(* Schneider Machine Expert - Basic project magnetic-pulse-modbus, file version 2.5.0.0 *)
(* ProjectInformations: Name=AGM1-lower *)
(* UserInformations: LastName=Aleksandr, FirstName=Kolodkin, PhoneNumber=+380963724869, CellNumber=+380996102231, Email=alexandr.kolodkin@gmail.com *)

HARDWARE
  Cpu 0: TM221CE40T
  EthernetConfiguration: NetworkName=M221, IpAllocationMode=FixedAddress, IpAddress=192.168.10.21, SubnetMask=255.255.255.0
  SerialLineConfiguration: Baud=Baud19200, Parity=ParityEven, DataBits=DataBits8, StopBits=StopBits1, PhysicalMedium=PhysicalMediumRs485, TransmissionMode=TransmissionModeModbusRtu, SlaveId=1, Addressing=SlaveAddressing
  MastTask: UsePeriodScanMode=false, PeriodScan=100
  FastTask: Period=255
  CpuBehavior: StartingMode=StartInRun, AutoSaveRamOnEeprom=true, WatchdogPeriod=250

SYMBOLS  (address, symbol, comment, settings)
  %M0       INPUT_0  "Дискретный вход #0"
  %M1       INPUT_1  "Дискретный вход #1"
  %M2       INPUT_2  "Дискретный вход #2"
  %M3       INPUT_3  "Дискретный вход #3"
  %M4       INPUT_4  "Дискретный вход #4"
  %M5       INPUT_5  "Дискретный вход #5"
  %M6       INPUT_6  "Дискретный вход #6"
  %M7       INPUT_7  "Дискретный вход #7"
  %M8       INPUT_8  "Дискретный вход #8"
  %M9       INPUT_9  "Дискретный вход #9"
  %M10      INPUT_10  "Дискретный вход #10"
  %M11      INPUT_11  "Дискретный вход #11"
  %M12      INPUT_12  "Дискретный вход #12"
  %M13      INPUT_13  "Дискретный вход #13"
  %M14      INPUT_14  "Дискретный вход #14"
  %M15      INPUT_15  "Дискретный вход #15"
  %M16      INPUT_16  "Дискретный вход #16"
  %M17      INPUT_17  "Дискретный вход #17"
  %M18      INPUT_18  "Дискретный вход #18"
  %M19      INPUT_19  "Дискретный вход #19"
  %M20      INPUT_20  "Дискретный вход #20"
  %M21      INPUT_21  "Дискретный вход #21"
  %M22      INPUT_22  "Дискретный вход #22"
  %M23      INPUT_23  "Дискретный вход #23"
  %M24      INPUT_24  "Дискретный вход модуля расширения #0"
  %M25      INPUT_25  "Дискретный вход модуля расширения #1"
  %M26      INPUT_26  "Дискретный вход модуля расширения #2"
  %M27      INPUT_27  "Дискретный вход модуля расширения #3"
  %M28      INPUT_28  "Дискретный вход модуля расширения #4"
  %M29      INPUT_29  "Дискретный вход модуля расширения #5"
  %M30      INPUT_30  "Дискретный вход модуля расширения #6"
  %M31      INPUT_31  "Дискретный вход модуля расширения #7"
  %M32      LOCAL_1  "Местный запуск обрушения 1-го бункера"
  %M33      LOCAL_2  "Местный запуск обрушения 2-го бункера"
  %M34      LOCAL_3  "Местный запуск обрушения 3-го бункера"
  %M35      LOCAL_4  "Местный запуск обрушения 4-го бункера"
  %M36      LOCAL_5  "Местный запуск обрушения 5-го бункера"
  %M37      LOCAL_6  "Местный запуск обрушения 6-го бункера"
  %M38      LOCAL_7  "Местный запуск обрушения 7-го бункера"
  %M39      LOCAL_8  "Местный запуск обрушения 8-го бункера"
  %M40      LOCAL_9  "Местный запуск обрушения 9-го бункера"
  %M41      LOCAL_10  "Местный запуск обрушения 10-го бункера"
  %M48      REMOTE_1  "Дистанционный запуск обрушения 1-го бункера"
  %M49      REMOTE_2  "Дистанционный запуск обрушения 2-го бункера"
  %M50      REMOTE_3  "Дистанционный запуск обрушения 3-го бункера"
  %M51      REMOTE_4  "Дистанционный запуск обрушения 4-го бункера"
  %M52      REMOTE_5  "Дистанционный запуск обрушения 5-го бункера"
  %M53      REMOTE_6  "Дистанционный запуск обрушения 6-го бункера"
  %M54      REMOTE_7  "Дистанционный запуск обрушения 7-го бункера"
  %M55      REMOTE_8  "Дистанционный запуск обрушения 8-го бункера"
  %M56      REMOTE_9  "Дистанционный запуск обрушения 9-го бункера"
  %M57      REMOTE_10  "Дистанционный запуск обрушения 10-го бункера"
  %M64      CMD_1  "Заказано обрушение 1-го бункера"
  %M65      CMD_2  "Заказано обрушение 2-го бункера"
  %M66      CMD_3  "Заказано обрушение 3-го бункера"
  %M67      CMD_4  "Заказано обрушение 4-го бункера"
  %M68      CMD_5  "Заказано обрушение 5-го бункера"
  %M69      CMD_6  "Заказано обрушение 6-го бункера"
  %M70      CMD_7  "Заказано обрушение 7-го бункера"
  %M71      CMD_8  "Заказано обрушение 8-го бункера"
  %M72      CMD_9  "Заказано обрушение 9-го бункера"
  %M73      CMD_10  "Заказано обрушение 10-го бункера"
  %M80      CMD  "Есть заказ на обрушение бункера"
  %M81      RESET  "Сброс"
  %M82      READY  "Готовность"
  %M83      FAULT  "Авария при заряде конденсатора"
  %M84      TEMP  "Промежуточная переменная для получения сигнала NEXT"
  %M85      PULSE  "Импульс"
  %M86      NEXT  "Переход к следующему заказу или завершение работы"
  %M87      CHARGED  "Конденсатор заряжен"
  %M88      LOCAL  "Выбрано местное управление"
  %M89      REMOTE  "Выбрано дистанционное управление"
  %M90      POWER  "Питание подано"
  %M91      CHARGE  "Комманда на заряд конденсатора"
  %M96      PULSE_1  "Запуск обрушения 1-го бункера"
  %M97      PULSE_2  "Запуск обрушения 2-го бункера"
  %M98      PULSE_3  "Запуск обрушения 3-го бункера"
  %M99      PULSE_4  "Запуск обрушения 4-го бункера"
  %M100     PULSE_5  "Запуск обрушения 5-го бункера"
  %M101     PULSE_6  "Запуск обрушения 6-го бункера"
  %M102     PULSE_7  "Запуск обрушения 7-го бункера"
  %M103     PULSE_8  "Запуск обрушения 8-го бункера"
  %M104     PULSE_9  "Запуск обрушения 9-го бункера"
  %M105     PULSE_10  "Запуск обрушения 10-го бункера"
  %M112     SELECTED_1  "Выполняется обрушение 1-го бункера"
  %M113     SELECTED_2  "Выполняется обрушение 2-го бункера"
  %M114     SELECTED_3  "Выполняется обрушение 3-го бункера"
  %M115     SELECTED_4  "Выполняется обрушение 4-го бункера"
  %M116     SELECTED_5  "Выполняется обрушение 5-го бункера"
  %M117     SELECTED_6  "Выполняется обрушение 6-го бункера"
  %M118     SELECTED_7  "Выполняется обрушение 7-го бункера"
  %M119     SELECTED_8  "Выполняется обрушение 8-го бункера"
  %M120     SELECTED_9  "Выполняется обрушение 9-го бункера"
  %M121     SELECTED_10  "Выполняется обрушение 10-го бункера"
  %M128     MODBUS_1  "Запуск обрушения 1-го бункера через ModBus"
  %M129     MODBUS_2  "Запуск обрушения 2-го бункера через ModBus"
  %M130     MODBUS_3  "Запуск обрушения 3-го бункера через ModBus"
  %M131     MODBUS_4  "Запуск обрушения 4-го бункера через ModBus"
  %M132     MODBUS_5  "Запуск обрушения 5-го бункера через ModBus"
  %M133     MODBUS_6  "Запуск обрушения 6-го бункера через ModBus"
  %M134     MODBUS_7  "Запуск обрушения 7-го бункера через ModBus"
  %M135     MODBUS_8  "Запуск обрушения 8-го бункера через ModBus"
  %M136     MODBUS_9  "Запуск обрушения 9-го бункера через ModBus"
  %M137     MODBUS_10  "Запуск обрушения 10-го бункера через ModBus"
  %M144     MODBUS  "Управление по сети ModBus"
  %M145     CHARGED_M  "Имитация конденсатора при управлении по ModBus'у"
  %M146     RESET_M  "Сброс аварии по сети ModBus"
  %M160     FAULT_1  "Сбой при обрушении 1-го бункера"
  %M161     FAULT_2  "Сбой при обрушении 2-го бункера"
  %M162     FAULT_3  "Сбой при обрушении 3-го бункера"
  %M163     FAULT_4  "Сбой при обрушении 4-го бункера"
  %M164     FAULT_5  "Сбой при обрушении 5-го бункера"
  %M165     FAULT_6  "Сбой при обрушении 6-го бункера"
  %M166     FAULT_7  "Сбой при обрушении 7-го бункера"
  %M167     FAULT_8  "Сбой при обрушении 8-го бункера"
  %M168     FAULT_9  "Сбой при обрушении 9-го бункера"
  %M169     FAULT_10  "Сбой при обрушении 10-го бункера"
  %TM0      READY_T  "Задержка готовности"  [Preset=10, Base=OneHundredMilliSeconds]
  %TM1      RESET_T  "Импульс сброса"  [Type=TOF, Preset=5, Base=OneHundredMilliSeconds]
  %TM2      CHARGE_T  "Задержка начала заряда конденсатора"  [Preset=10, Base=TenMilliSeconds]
  %TM3      CHARGE_FAULT_T  "Задержка до аварии: конденсатор не заряжен"  [Preset=15, Base=OneSecond]
  %TM4      DISCHARGE_FAULT_T  "Задержка до аварии: конденсатор не разряжен"  [Preset=30, Base=OneHundredMilliSeconds]
  %TM5      PULSE_START_T  "Задержка перед подачей импульса"  [Preset=20, Base=OneHundredMilliSeconds]
  %TM6      PULSE_T  "Продолжительность импульса"  [Type=TP, Preset=50, Base=TenMilliSeconds]
  %TM7      NEXT_T  "Задержка перед началом проверки (должно быть меньше чем DISCHARGE_FAULT_T)"  [Type=TOF, Preset=5, Base=OneHundredMilliSeconds]
  %TM10     CMD1_T  "Формирование имульса заказа #1"  [Type=TP, Preset=1, Base=TenMilliSeconds]
  %TM11     CMD2_T  "Формирование имульса заказа #2"  [Type=TP, Preset=1, Base=TenMilliSeconds]
  %TM12     CMD3_T  "Формирование имульса заказа #3"  [Type=TP, Preset=1, Base=TenMilliSeconds]
  %TM13     CMD4_T  "Формирование имульса заказа #4"  [Type=TP, Preset=1, Base=TenMilliSeconds]
  %TM14     CMD5_T  "Формирование имульса заказа #5"  [Type=TP, Preset=1, Base=TenMilliSeconds]
  %TM15     CMD6_T  "Формирование имульса заказа #6"  [Type=TP, Preset=1, Base=TenMilliSeconds]
  %TM16     CMD7_T  "Формирование имульса заказа #7"  [Type=TP, Preset=1, Base=TenMilliSeconds]
  %TM17     CMD8_T  "Формирование имульса заказа #8"  [Type=TP, Preset=1, Base=TenMilliSeconds]
  %READ_VAR0 RD3_1  [Link(Value(FBComLinkParameterEnums=SerialLine1)), RemoteDeviceId(Value(int=1)), Timeout(Value(int=100)), ObjType(Value(FBComObjTypeParameterEnums=MW)), FirstObj(Value(int=0)), Quantity(Value(int=16)), IndexData(Value(int=0))]
  %I0.0     IN_0
  %I0.1     IN_1
  %I0.2     IN_2
  %I0.3     IN_3
  %I0.4     IN_4
  %I0.5     IN_5
  %I0.6     IN_6
  %I0.7     IN_7
  %I0.8     IN_8
  %I0.9     IN_9
  %I0.10    IN_10
  %I0.11    IN_11
  %I0.12    IN_12
  %I0.13    IN_13
  %I0.14    IN_14
  %I0.15    IN_15
  %I0.16    IN_16
  %I0.17    IN_17
  %I0.18    IN_18
  %I0.19    IN_19
  %I0.20    IN_20
  %I0.21    IN_21
  %I0.22    IN_22
  %I0.23    IN_23
  %Q0.0     OUTPUT_0
  %Q0.1     OUTPUT_1  "Запуск №2"
  %Q0.2     OUTPUT_2  "Запуск №3"
  %Q0.3     OUTPUT_3  "Запуск №4"
  %Q0.4     OUTPUT_4  "Запуск №5"
  %Q0.5     OUTPUT_5  "Запуск №6"
  %Q0.6     OUTPUT_6  "Запуск №7"
  %Q0.7     OUTPUT_7  "Запуск №8"
  %Q0.8     OUTPUT_8
  %Q0.9     OUTPUT_9
  %Q0.10    OUTPUT_10  "Готовность"
  %Q0.11    OUTPUT_11
  %Q0.12    OUTPUT_12
  %Q0.13    OUTPUT_13
  %Q0.14    OUTPUT_14  "Включить заряд конденсатора"
  %Q0.15    OUTPUT_15  "Ошибка"

POU Main logic
  (* SectionNumber=1 *)

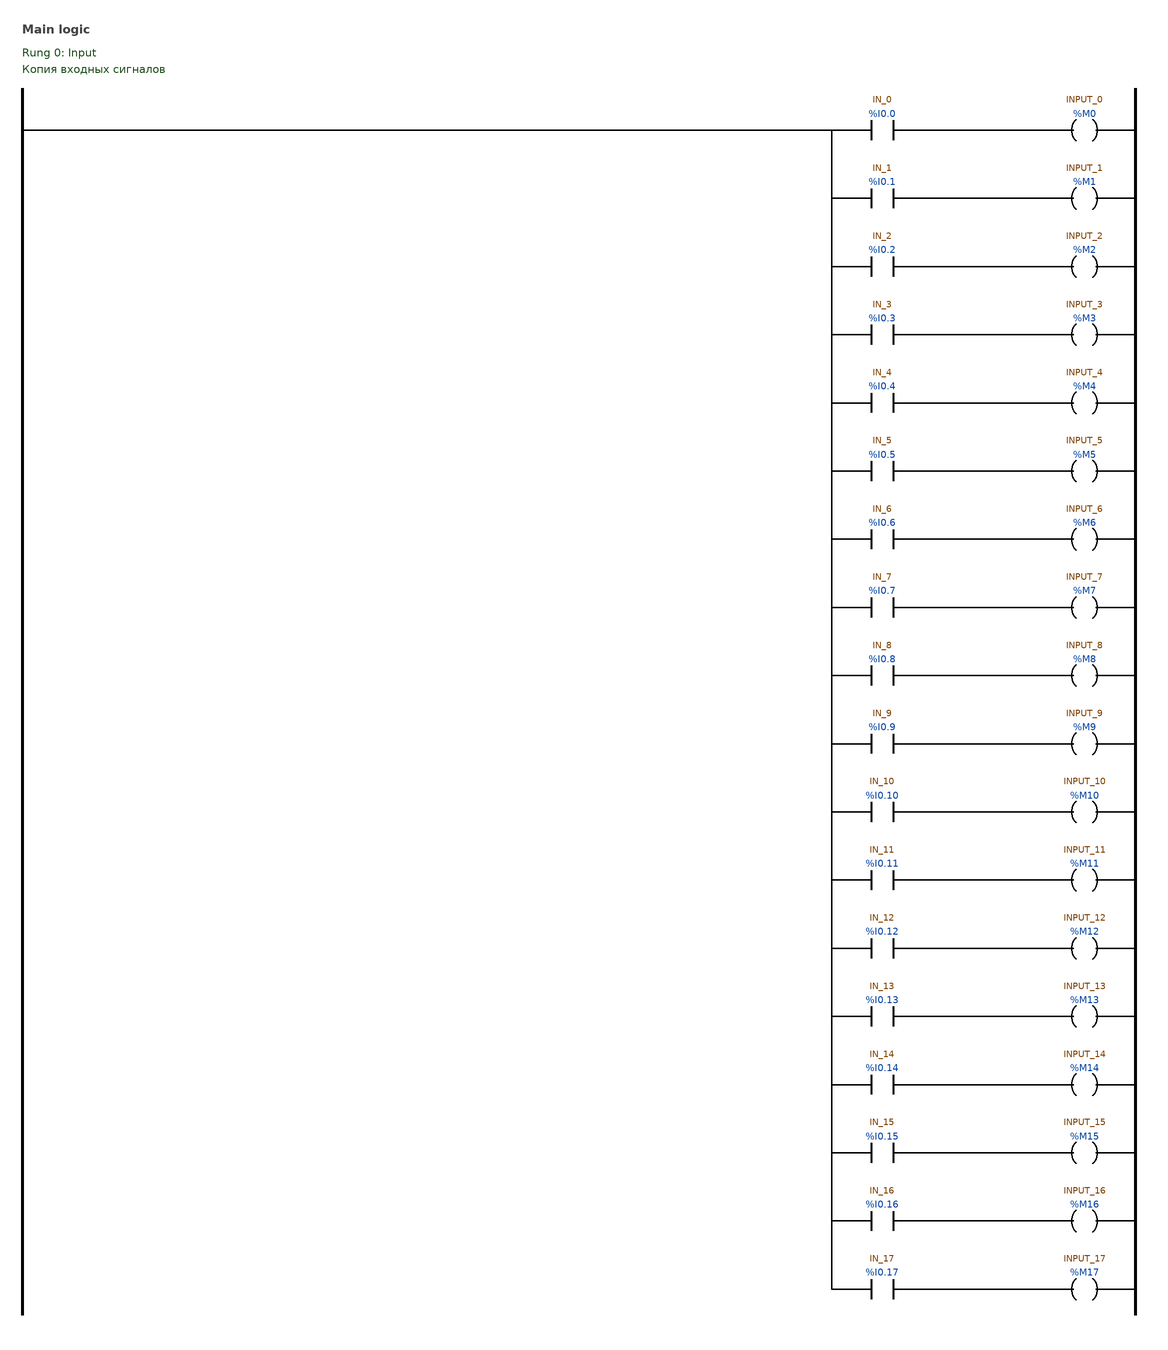

// Rung 0: Input
// Копия входных сигналов
  LD 1
  MPS
  AND %I0.0               (* IN_0 *)
  ST %M0                  (* INPUT_0 *)
  MRD
  AND %I0.1               (* IN_1 *)
  ST %M1                  (* INPUT_1 *)
  MRD
  AND %I0.2               (* IN_2 *)
  ST %M2                  (* INPUT_2 *)
  MRD
  AND %I0.3               (* IN_3 *)
  ST %M3                  (* INPUT_3 *)
  MRD
  AND %I0.4               (* IN_4 *)
  ST %M4                  (* INPUT_4 *)
  MRD
  AND %I0.5               (* IN_5 *)
  ST %M5                  (* INPUT_5 *)
  MRD
  AND %I0.6               (* IN_6 *)
  ST %M6                  (* INPUT_6 *)
  MRD
  AND %I0.7               (* IN_7 *)
  ST %M7                  (* INPUT_7 *)
  MRD
  AND %I0.8               (* IN_8 *)
  ST %M8                  (* INPUT_8 *)
  MRD
  AND %I0.9               (* IN_9 *)
  ST %M9                  (* INPUT_9 *)
  MRD
  AND %I0.10              (* IN_10 *)
  ST %M10                 (* INPUT_10 *)
  MRD
  AND %I0.11              (* IN_11 *)
  ST %M11                 (* INPUT_11 *)
  MRD
  AND %I0.12              (* IN_12 *)
  ST %M12                 (* INPUT_12 *)
  MRD
  AND %I0.13              (* IN_13 *)
  ST %M13                 (* INPUT_13 *)
  MRD
  AND %I0.14              (* IN_14 *)
  ST %M14                 (* INPUT_14 *)
  MRD
  AND %I0.15              (* IN_15 *)
  ST %M15                 (* INPUT_15 *)
  MRD
  AND %I0.16              (* IN_16 *)
  ST %M16                 (* INPUT_16 *)
  MPP
  AND %I0.17              (* IN_17 *)
  ST %M17                 (* INPUT_17 *)
  // as ST:
  //   INPUT_0 := IN_0;
  //   INPUT_1 := IN_1;
  //   INPUT_2 := IN_2;
  //   INPUT_3 := IN_3;
  //   INPUT_4 := IN_4;
  //   INPUT_5 := IN_5;
  //   INPUT_6 := IN_6;
  //   INPUT_7 := IN_7;
  //   INPUT_8 := IN_8;
  //   INPUT_9 := IN_9;
  //   INPUT_10 := IN_10;
  //   INPUT_11 := IN_11;
  //   INPUT_12 := IN_12;
  //   INPUT_13 := IN_13;
  //   INPUT_14 := IN_14;
  //   INPUT_15 := IN_15;
  //   INPUT_16 := IN_16;
  //   INPUT_17 := IN_17;

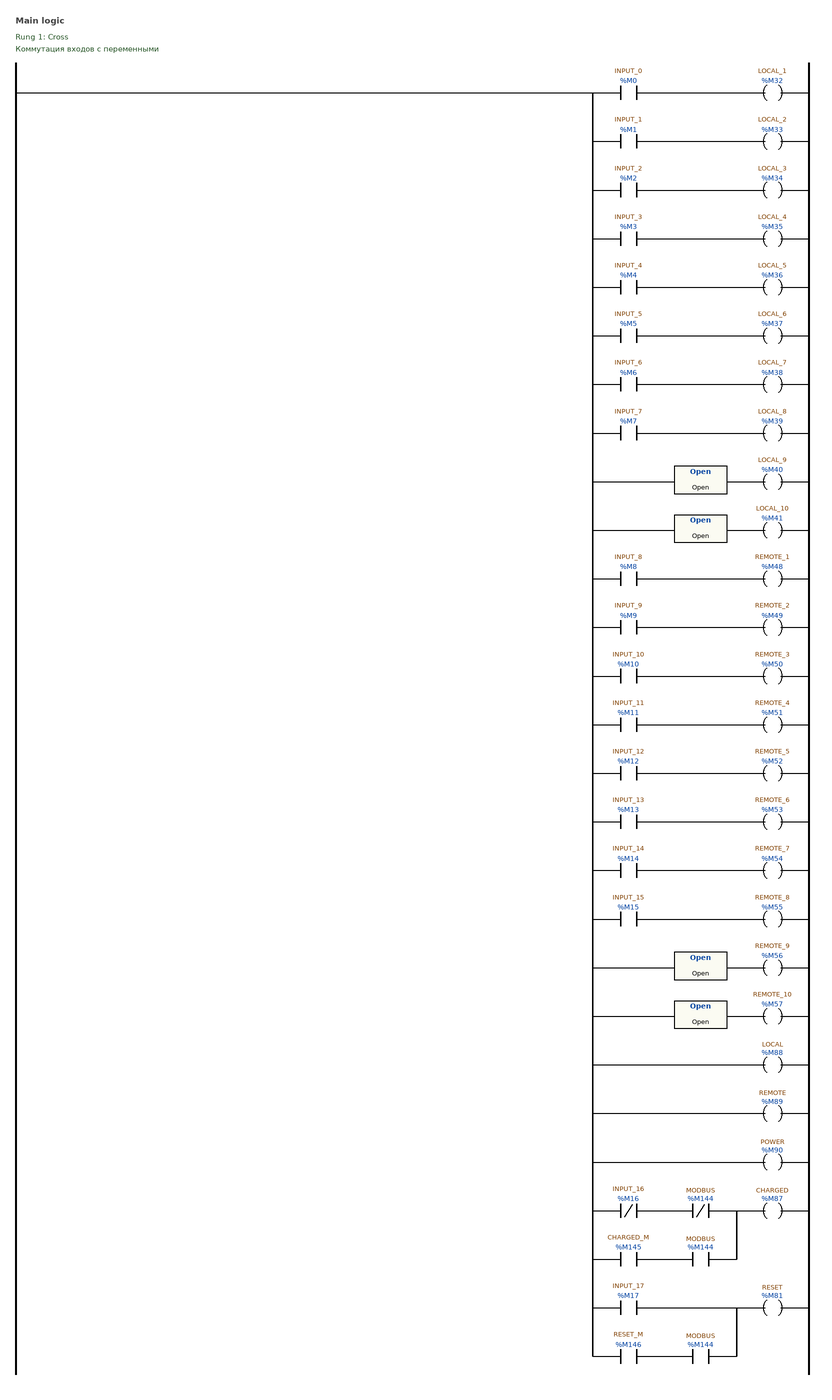

// Rung 1: Cross
// Коммутация входов с переменными
  LD 1
  MPS
  AND %M0                 (* INPUT_0 *)
  ST %M32                 (* LOCAL_1 *)
  MRD
  AND %M1                 (* INPUT_1 *)
  ST %M33                 (* LOCAL_2 *)
  MRD
  AND %M2                 (* INPUT_2 *)
  ST %M34                 (* LOCAL_3 *)
  MRD
  AND %M3                 (* INPUT_3 *)
  ST %M35                 (* LOCAL_4 *)
  MRD
  AND %M4                 (* INPUT_4 *)
  ST %M36                 (* LOCAL_5 *)
  MRD
  AND %M5                 (* INPUT_5 *)
  ST %M37                 (* LOCAL_6 *)
  MRD
  AND %M6                 (* INPUT_6 *)
  ST %M38                 (* LOCAL_7 *)
  MRD
  AND %M7                 (* INPUT_7 *)
  ST %M39                 (* LOCAL_8 *)
  MRD
  AND 0
  ST %M40                 (* LOCAL_9 *)
  MRD
  AND 0
  ST %M41                 (* LOCAL_10 *)
  MRD
  AND %M8                 (* INPUT_8 *)
  ST %M48                 (* REMOTE_1 *)
  MRD
  AND %M9                 (* INPUT_9 *)
  ST %M49                 (* REMOTE_2 *)
  MRD
  AND %M10                (* INPUT_10 *)
  ST %M50                 (* REMOTE_3 *)
  MRD
  AND %M11                (* INPUT_11 *)
  ST %M51                 (* REMOTE_4 *)
  MRD
  AND %M12                (* INPUT_12 *)
  ST %M52                 (* REMOTE_5 *)
  MRD
  AND %M13                (* INPUT_13 *)
  ST %M53                 (* REMOTE_6 *)
  MRD
  AND %M14                (* INPUT_14 *)
  ST %M54                 (* REMOTE_7 *)
  MRD
  AND %M15                (* INPUT_15 *)
  ST %M55                 (* REMOTE_8 *)
  MRD
  AND 0
  ST %M56                 (* REMOTE_9 *)
  MRD
  AND 0
  ST %M57                 (* REMOTE_10 *)
  MRD
  AND 1
  ST %M88                 (* LOCAL *)
  MRD
  AND 1
  ST %M89                 (* REMOTE *)
  MRD
  AND 1
  ST %M90                 (* POWER *)
  MRD
  AND(N %M16              (* INPUT_16 *)
  ANDN %M144              (* MODBUS *)
  OR( %M145               (* CHARGED_M *)
  AND %M144               (* MODBUS *)
  )
  )
  ST %M87                 (* CHARGED *)
  MPP
  AND( %M17               (* INPUT_17 *)
  OR( %M146               (* RESET_M *)
  AND %M144               (* MODBUS *)
  )
  )
  ST %M81                 (* RESET *)
  // as ST:
  //   LOCAL_1 := INPUT_0;
  //   LOCAL_2 := INPUT_1;
  //   LOCAL_3 := INPUT_2;
  //   LOCAL_4 := INPUT_3;
  //   LOCAL_5 := INPUT_4;
  //   LOCAL_6 := INPUT_5;
  //   LOCAL_7 := INPUT_6;
  //   LOCAL_8 := INPUT_7;
  //   LOCAL_9 := FALSE;
  //   LOCAL_10 := FALSE;
  //   REMOTE_1 := INPUT_8;
  //   REMOTE_2 := INPUT_9;
  //   REMOTE_3 := INPUT_10;
  //   REMOTE_4 := INPUT_11;
  //   REMOTE_5 := INPUT_12;
  //   REMOTE_6 := INPUT_13;
  //   REMOTE_7 := INPUT_14;
  //   REMOTE_8 := INPUT_15;
  //   REMOTE_9 := FALSE;
  //   REMOTE_10 := FALSE;
  //   LOCAL := TRUE;
  //   REMOTE := TRUE;
  //   POWER := TRUE;
  //   CHARGED := NOT INPUT_16 AND NOT MODBUS OR CHARGED_M AND MODBUS;
  //   RESET := INPUT_17 OR RESET_M AND MODBUS;

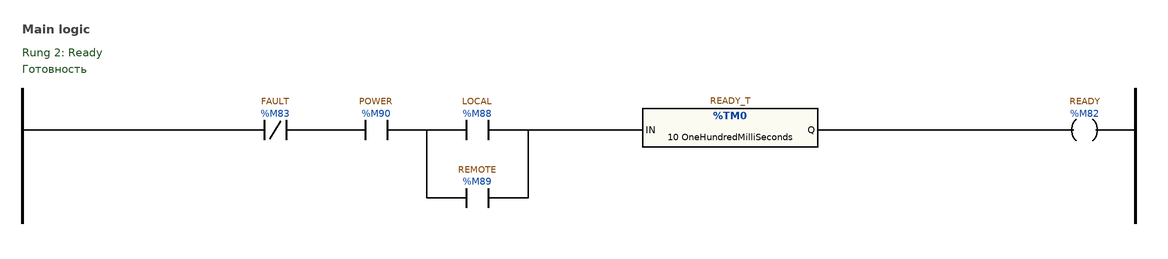

// Rung 2: Ready
// Готовность
  BLK %TM0                (* READY_T *)
  LDN %M83                (* FAULT *)
  AND %M90                (* POWER *)
  AND( %M88               (* LOCAL *)
  OR %M89                 (* REMOTE *)
  )
  IN
  OUT_BLK
  LD Q
  ST %M82                 (* READY *)
  END_BLK
  // as ST:
  //   READY_T(IN := NOT FAULT AND POWER AND (LOCAL OR REMOTE));
  //   READY := READY_T.Q;

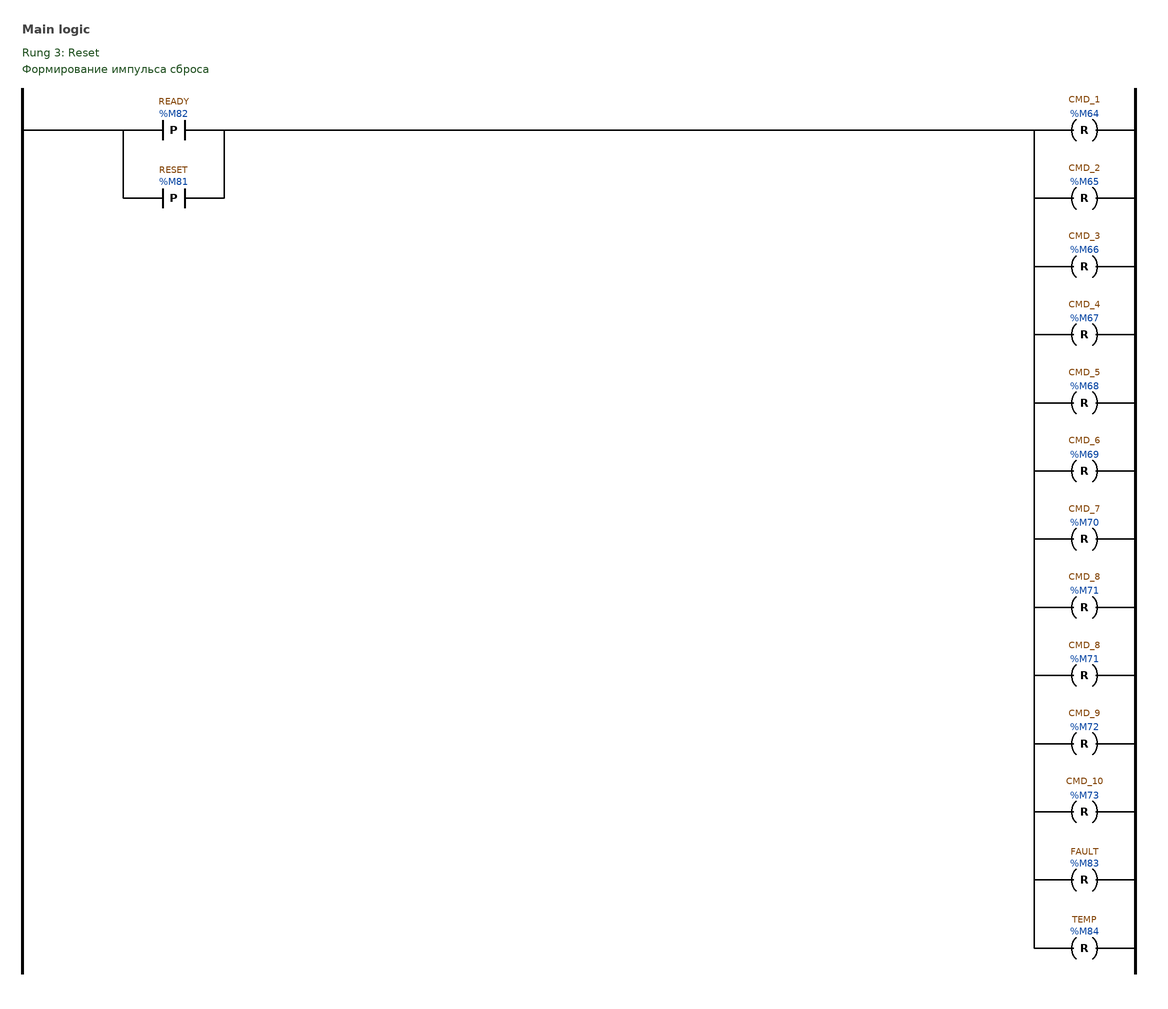

// Rung 3: Reset
// Формирование импульса сброса
  LD 1
  AND(R %M82              (* READY *)
  ORR %M81                (* RESET *)
  )
  R %M64                  (* CMD_1 *)
  R %M65                  (* CMD_2 *)
  R %M66                  (* CMD_3 *)
  R %M67                  (* CMD_4 *)
  R %M68                  (* CMD_5 *)
  R %M69                  (* CMD_6 *)
  R %M70                  (* CMD_7 *)
  R %M71                  (* CMD_8 *)
  R %M71                  (* CMD_8 *)
  R %M72                  (* CMD_9 *)
  R %M73                  (* CMD_10 *)
  R %M83                  (* FAULT *)
  R %M84                  (* TEMP *)
  // as ST:
  //   IF RISING(READY) OR RISING(RESET) THEN CMD_1 := FALSE; END_IF;
  //   IF RISING(READY) OR RISING(RESET) THEN CMD_2 := FALSE; END_IF;
  //   IF RISING(READY) OR RISING(RESET) THEN CMD_3 := FALSE; END_IF;
  //   IF RISING(READY) OR RISING(RESET) THEN CMD_4 := FALSE; END_IF;
  //   IF RISING(READY) OR RISING(RESET) THEN CMD_5 := FALSE; END_IF;
  //   IF RISING(READY) OR RISING(RESET) THEN CMD_6 := FALSE; END_IF;
  //   IF RISING(READY) OR RISING(RESET) THEN CMD_7 := FALSE; END_IF;
  //   IF RISING(READY) OR RISING(RESET) THEN CMD_8 := FALSE; END_IF;
  //   IF RISING(READY) OR RISING(RESET) THEN CMD_8 := FALSE; END_IF;
  //   IF RISING(READY) OR RISING(RESET) THEN CMD_9 := FALSE; END_IF;
  //   IF RISING(READY) OR RISING(RESET) THEN CMD_10 := FALSE; END_IF;
  //   IF RISING(READY) OR RISING(RESET) THEN FAULT := FALSE; END_IF;
  //   IF RISING(READY) OR RISING(RESET) THEN TEMP := FALSE; END_IF;

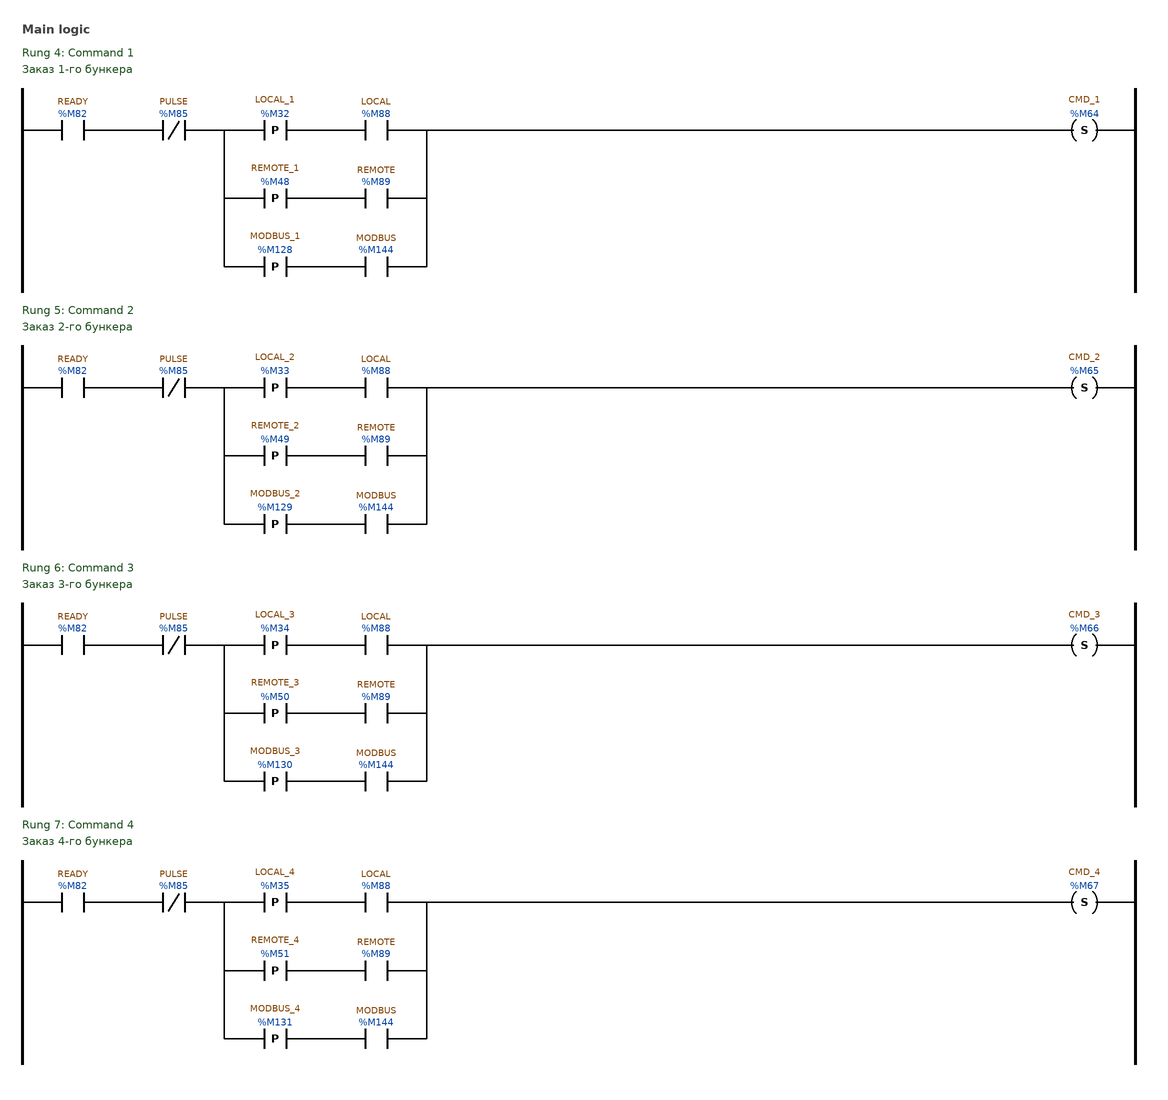

// Rung 4: Command 1
// Заказ 1-го бункера
  LD %M82                 (* READY *)
  ANDN %M85               (* PULSE *)
  AND(R %M32              (* LOCAL_1 *)
  AND %M88                (* LOCAL *)
  OR(R %M48               (* REMOTE_1 *)
  AND %M89                (* REMOTE *)
  )
  OR(R %M128              (* MODBUS_1 *)
  AND %M144               (* MODBUS *)
  )
  )
  S %M64                  (* CMD_1 *)
  // as ST:
  //   IF READY AND NOT PULSE AND (RISING(LOCAL_1) AND LOCAL OR RISING(REMOTE_1) AND REMOTE OR RISING(MODBUS_1) AND MODBUS) THEN CMD_1 := TRUE; END_IF;

// Rung 5: Command 2
// Заказ 2-го бункера
  LD %M82                 (* READY *)
  ANDN %M85               (* PULSE *)
  AND(R %M33              (* LOCAL_2 *)
  AND %M88                (* LOCAL *)
  OR(R %M49               (* REMOTE_2 *)
  AND %M89                (* REMOTE *)
  )
  OR(R %M129              (* MODBUS_2 *)
  AND %M144               (* MODBUS *)
  )
  )
  S %M65                  (* CMD_2 *)
  // as ST:
  //   IF READY AND NOT PULSE AND (RISING(LOCAL_2) AND LOCAL OR RISING(REMOTE_2) AND REMOTE OR RISING(MODBUS_2) AND MODBUS) THEN CMD_2 := TRUE; END_IF;

// Rung 6: Command 3
// Заказ 3-го бункера
  LD %M82                 (* READY *)
  ANDN %M85               (* PULSE *)
  AND(R %M34              (* LOCAL_3 *)
  AND %M88                (* LOCAL *)
  OR(R %M50               (* REMOTE_3 *)
  AND %M89                (* REMOTE *)
  )
  OR(R %M130              (* MODBUS_3 *)
  AND %M144               (* MODBUS *)
  )
  )
  S %M66                  (* CMD_3 *)
  // as ST:
  //   IF READY AND NOT PULSE AND (RISING(LOCAL_3) AND LOCAL OR RISING(REMOTE_3) AND REMOTE OR RISING(MODBUS_3) AND MODBUS) THEN CMD_3 := TRUE; END_IF;

// Rung 7: Command 4
// Заказ 4-го бункера
  LD %M82                 (* READY *)
  ANDN %M85               (* PULSE *)
  AND(R %M35              (* LOCAL_4 *)
  AND %M88                (* LOCAL *)
  OR(R %M51               (* REMOTE_4 *)
  AND %M89                (* REMOTE *)
  )
  OR(R %M131              (* MODBUS_4 *)
  AND %M144               (* MODBUS *)
  )
  )
  S %M67                  (* CMD_4 *)
  // as ST:
  //   IF READY AND NOT PULSE AND (RISING(LOCAL_4) AND LOCAL OR RISING(REMOTE_4) AND REMOTE OR RISING(MODBUS_4) AND MODBUS) THEN CMD_4 := TRUE; END_IF;

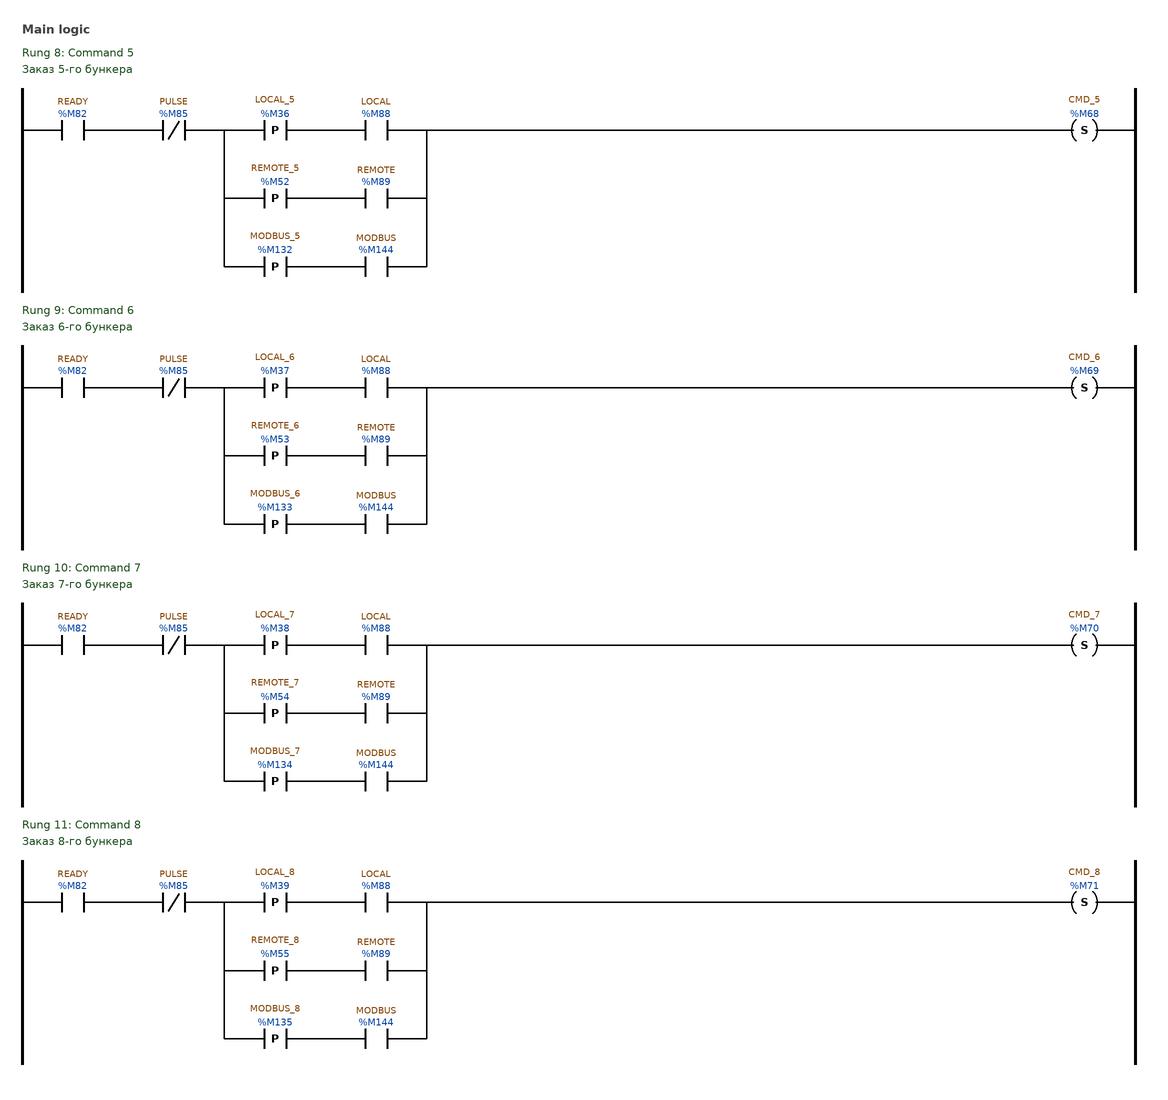

// Rung 8: Command 5
// Заказ 5-го бункера
  LD %M82                 (* READY *)
  ANDN %M85               (* PULSE *)
  AND(R %M36              (* LOCAL_5 *)
  AND %M88                (* LOCAL *)
  OR(R %M52               (* REMOTE_5 *)
  AND %M89                (* REMOTE *)
  )
  OR(R %M132              (* MODBUS_5 *)
  AND %M144               (* MODBUS *)
  )
  )
  S %M68                  (* CMD_5 *)
  // as ST:
  //   IF READY AND NOT PULSE AND (RISING(LOCAL_5) AND LOCAL OR RISING(REMOTE_5) AND REMOTE OR RISING(MODBUS_5) AND MODBUS) THEN CMD_5 := TRUE; END_IF;

// Rung 9: Command 6
// Заказ 6-го бункера
  LD %M82                 (* READY *)
  ANDN %M85               (* PULSE *)
  AND(R %M37              (* LOCAL_6 *)
  AND %M88                (* LOCAL *)
  OR(R %M53               (* REMOTE_6 *)
  AND %M89                (* REMOTE *)
  )
  OR(R %M133              (* MODBUS_6 *)
  AND %M144               (* MODBUS *)
  )
  )
  S %M69                  (* CMD_6 *)
  // as ST:
  //   IF READY AND NOT PULSE AND (RISING(LOCAL_6) AND LOCAL OR RISING(REMOTE_6) AND REMOTE OR RISING(MODBUS_6) AND MODBUS) THEN CMD_6 := TRUE; END_IF;

// Rung 10: Command 7
// Заказ 7-го бункера
  LD %M82                 (* READY *)
  ANDN %M85               (* PULSE *)
  AND(R %M38              (* LOCAL_7 *)
  AND %M88                (* LOCAL *)
  OR(R %M54               (* REMOTE_7 *)
  AND %M89                (* REMOTE *)
  )
  OR(R %M134              (* MODBUS_7 *)
  AND %M144               (* MODBUS *)
  )
  )
  S %M70                  (* CMD_7 *)
  // as ST:
  //   IF READY AND NOT PULSE AND (RISING(LOCAL_7) AND LOCAL OR RISING(REMOTE_7) AND REMOTE OR RISING(MODBUS_7) AND MODBUS) THEN CMD_7 := TRUE; END_IF;

// Rung 11: Command 8
// Заказ 8-го бункера
  LD %M82                 (* READY *)
  ANDN %M85               (* PULSE *)
  AND(R %M39              (* LOCAL_8 *)
  AND %M88                (* LOCAL *)
  OR(R %M55               (* REMOTE_8 *)
  AND %M89                (* REMOTE *)
  )
  OR(R %M135              (* MODBUS_8 *)
  AND %M144               (* MODBUS *)
  )
  )
  S %M71                  (* CMD_8 *)
  // as ST:
  //   IF READY AND NOT PULSE AND (RISING(LOCAL_8) AND LOCAL OR RISING(REMOTE_8) AND REMOTE OR RISING(MODBUS_8) AND MODBUS) THEN CMD_8 := TRUE; END_IF;

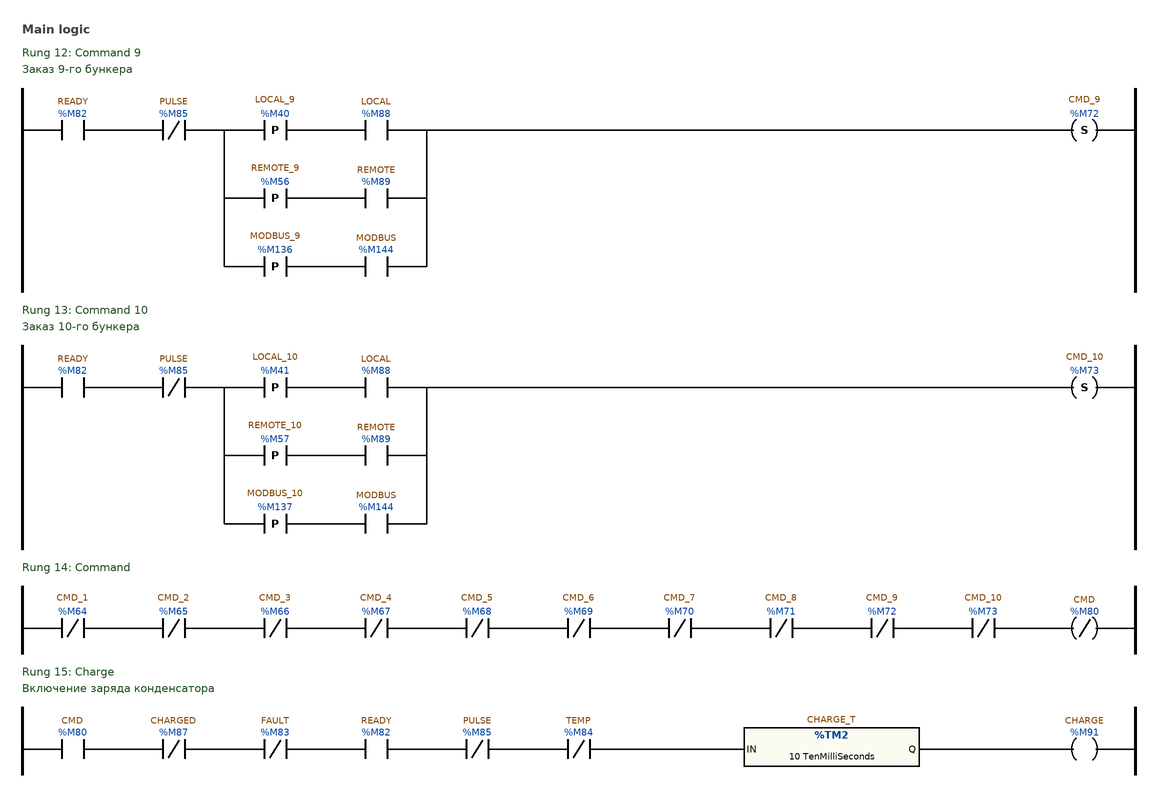

// Rung 12: Command 9
// Заказ 9-го бункера
  LD %M82                 (* READY *)
  ANDN %M85               (* PULSE *)
  AND(R %M40              (* LOCAL_9 *)
  AND %M88                (* LOCAL *)
  OR(R %M56               (* REMOTE_9 *)
  AND %M89                (* REMOTE *)
  )
  OR(R %M136              (* MODBUS_9 *)
  AND %M144               (* MODBUS *)
  )
  )
  S %M72                  (* CMD_9 *)
  // as ST:
  //   IF READY AND NOT PULSE AND (RISING(LOCAL_9) AND LOCAL OR RISING(REMOTE_9) AND REMOTE OR RISING(MODBUS_9) AND MODBUS) THEN CMD_9 := TRUE; END_IF;

// Rung 13: Command 10
// Заказ 10-го бункера
  LD %M82                 (* READY *)
  ANDN %M85               (* PULSE *)
  AND(R %M41              (* LOCAL_10 *)
  AND %M88                (* LOCAL *)
  OR(R %M57               (* REMOTE_10 *)
  AND %M89                (* REMOTE *)
  )
  OR(R %M137              (* MODBUS_10 *)
  AND %M144               (* MODBUS *)
  )
  )
  S %M73                  (* CMD_10 *)
  // as ST:
  //   IF READY AND NOT PULSE AND (RISING(LOCAL_10) AND LOCAL OR RISING(REMOTE_10) AND REMOTE OR RISING(MODBUS_10) AND MODBUS) THEN CMD_10 := TRUE; END_IF;

// Rung 14: Command
  LDN %M64                (* CMD_1 *)
  ANDN %M65               (* CMD_2 *)
  ANDN %M66               (* CMD_3 *)
  ANDN %M67               (* CMD_4 *)
  ANDN %M68               (* CMD_5 *)
  ANDN %M69               (* CMD_6 *)
  ANDN %M70               (* CMD_7 *)
  ANDN %M71               (* CMD_8 *)
  ANDN %M72               (* CMD_9 *)
  ANDN %M73               (* CMD_10 *)
  STN %M80                (* CMD *)
  // as ST:
  //   CMD := NOT (NOT CMD_1 AND NOT CMD_2 AND NOT CMD_3 AND NOT CMD_4 AND NOT CMD_5 AND NOT CMD_6 AND NOT CMD_7 AND NOT CMD_8 AND NOT CMD_9 AND NOT CMD_10);

// Rung 15: Charge
// Включение заряда конденсатора
  BLK %TM2                (* CHARGE_T *)
  LD %M80                 (* CMD *)
  ANDN %M87               (* CHARGED *)
  ANDN %M83               (* FAULT *)
  AND %M82                (* READY *)
  ANDN %M85               (* PULSE *)
  ANDN %M84               (* TEMP *)
  IN
  OUT_BLK
  LD Q
  ST %M91                 (* CHARGE *)
  END_BLK
  // as ST:
  //   CHARGE_T(IN := CMD AND NOT CHARGED AND NOT FAULT AND READY AND NOT PULSE AND NOT TEMP);
  //   CHARGE := CHARGE_T.Q;

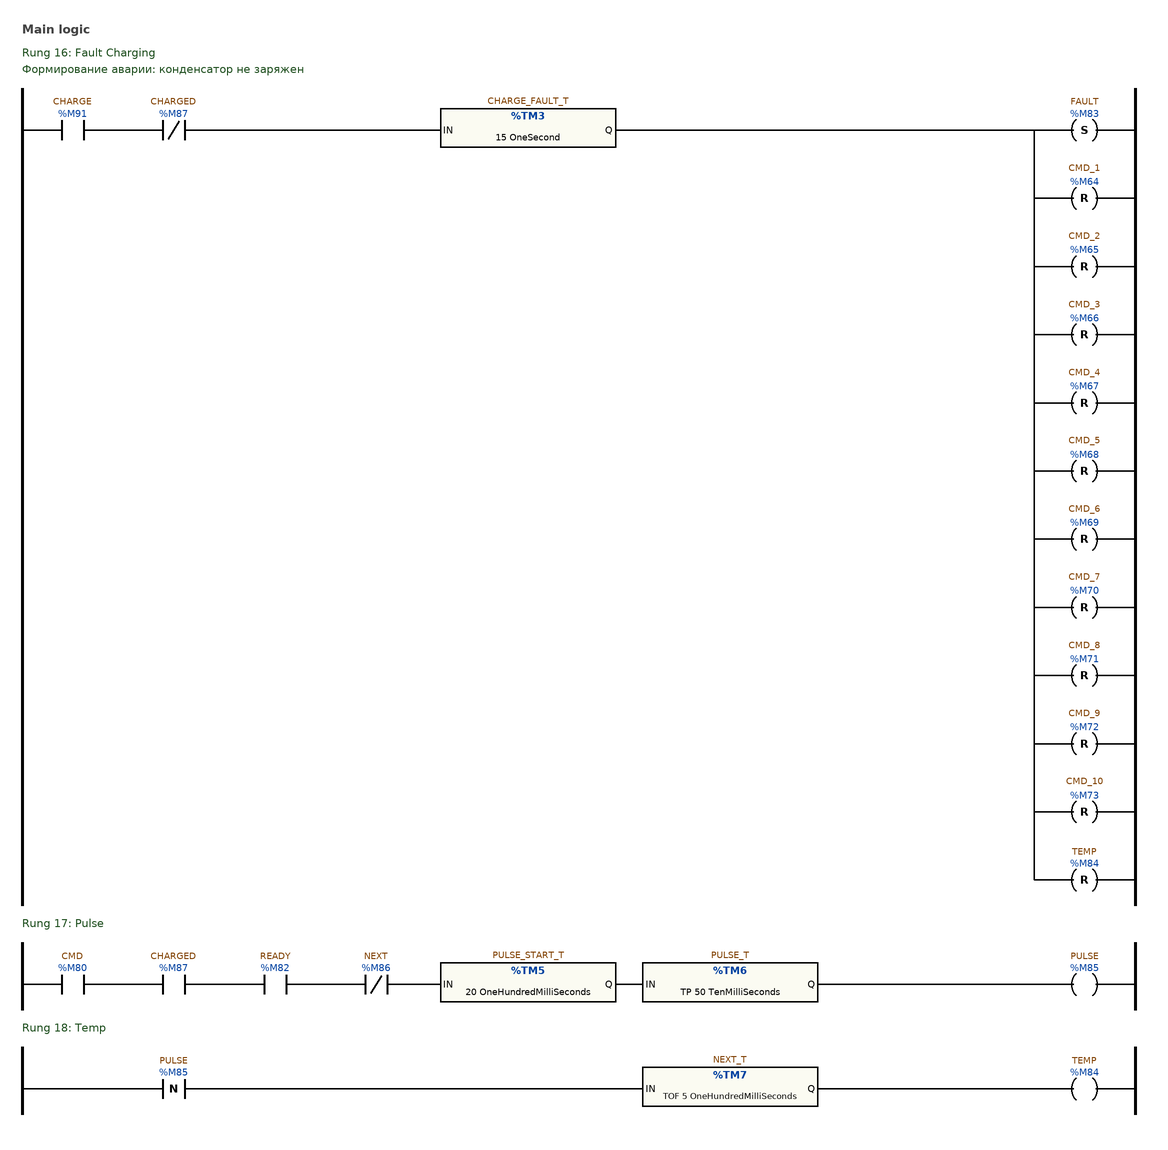

// Rung 16: Fault Charging
// Формирование аварии: конденсатор не заряжен
  BLK %TM3                (* CHARGE_FAULT_T *)
  LD %M91                 (* CHARGE *)
  ANDN %M87               (* CHARGED *)
  IN
  OUT_BLK
  LD Q
  S %M83                  (* FAULT *)
  R %M64                  (* CMD_1 *)
  R %M65                  (* CMD_2 *)
  R %M66                  (* CMD_3 *)
  R %M67                  (* CMD_4 *)
  R %M68                  (* CMD_5 *)
  R %M69                  (* CMD_6 *)
  R %M70                  (* CMD_7 *)
  R %M71                  (* CMD_8 *)
  R %M72                  (* CMD_9 *)
  R %M73                  (* CMD_10 *)
  R %M84                  (* TEMP *)
  END_BLK
  // as ST:
  //   CHARGE_FAULT_T(IN := CHARGE AND NOT CHARGED);
  //   IF CHARGE_FAULT_T.Q THEN FAULT := TRUE; END_IF;
  //   IF CHARGE_FAULT_T.Q THEN CMD_1 := FALSE; END_IF;
  //   IF CHARGE_FAULT_T.Q THEN CMD_2 := FALSE; END_IF;
  //   IF CHARGE_FAULT_T.Q THEN CMD_3 := FALSE; END_IF;
  //   IF CHARGE_FAULT_T.Q THEN CMD_4 := FALSE; END_IF;
  //   IF CHARGE_FAULT_T.Q THEN CMD_5 := FALSE; END_IF;
  //   IF CHARGE_FAULT_T.Q THEN CMD_6 := FALSE; END_IF;
  //   IF CHARGE_FAULT_T.Q THEN CMD_7 := FALSE; END_IF;
  //   IF CHARGE_FAULT_T.Q THEN CMD_8 := FALSE; END_IF;
  //   IF CHARGE_FAULT_T.Q THEN CMD_9 := FALSE; END_IF;
  //   IF CHARGE_FAULT_T.Q THEN CMD_10 := FALSE; END_IF;
  //   IF CHARGE_FAULT_T.Q THEN TEMP := FALSE; END_IF;

// Rung 17: Pulse
  LD 1
  MULTIFB
  BLK %TM5                (* PULSE_START_T *)
  LD %M80                 (* CMD *)
  AND %M87                (* CHARGED *)
  AND %M82                (* READY *)
  ANDN %M86               (* NEXT *)
  IN
  OUT_BLK
  LD Q
  ST %MW2000:X0
  END_BLK
  BLK %TM6                (* PULSE_T *)
  LD %MW2000:X0
  IN
  OUT_BLK
  LD Q
  ST %M85                 (* PULSE *)
  END_BLK
  MULTIFB
  // as ST:
  //   PULSE_START_T(IN := CMD AND CHARGED AND READY AND NOT NEXT);
  //   PULSE_T(IN := PULSE_START_T.Q);
  //   PULSE := PULSE_T.Q;

// Rung 18: Temp
  BLK %TM7                (* NEXT_T *)
  LDF %M85                (* PULSE *)
  IN
  OUT_BLK
  LD Q
  ST %M84                 (* TEMP *)
  END_BLK
  // as ST:
  //   NEXT_T(IN := FALLING(PULSE));
  //   TEMP := NEXT_T.Q;

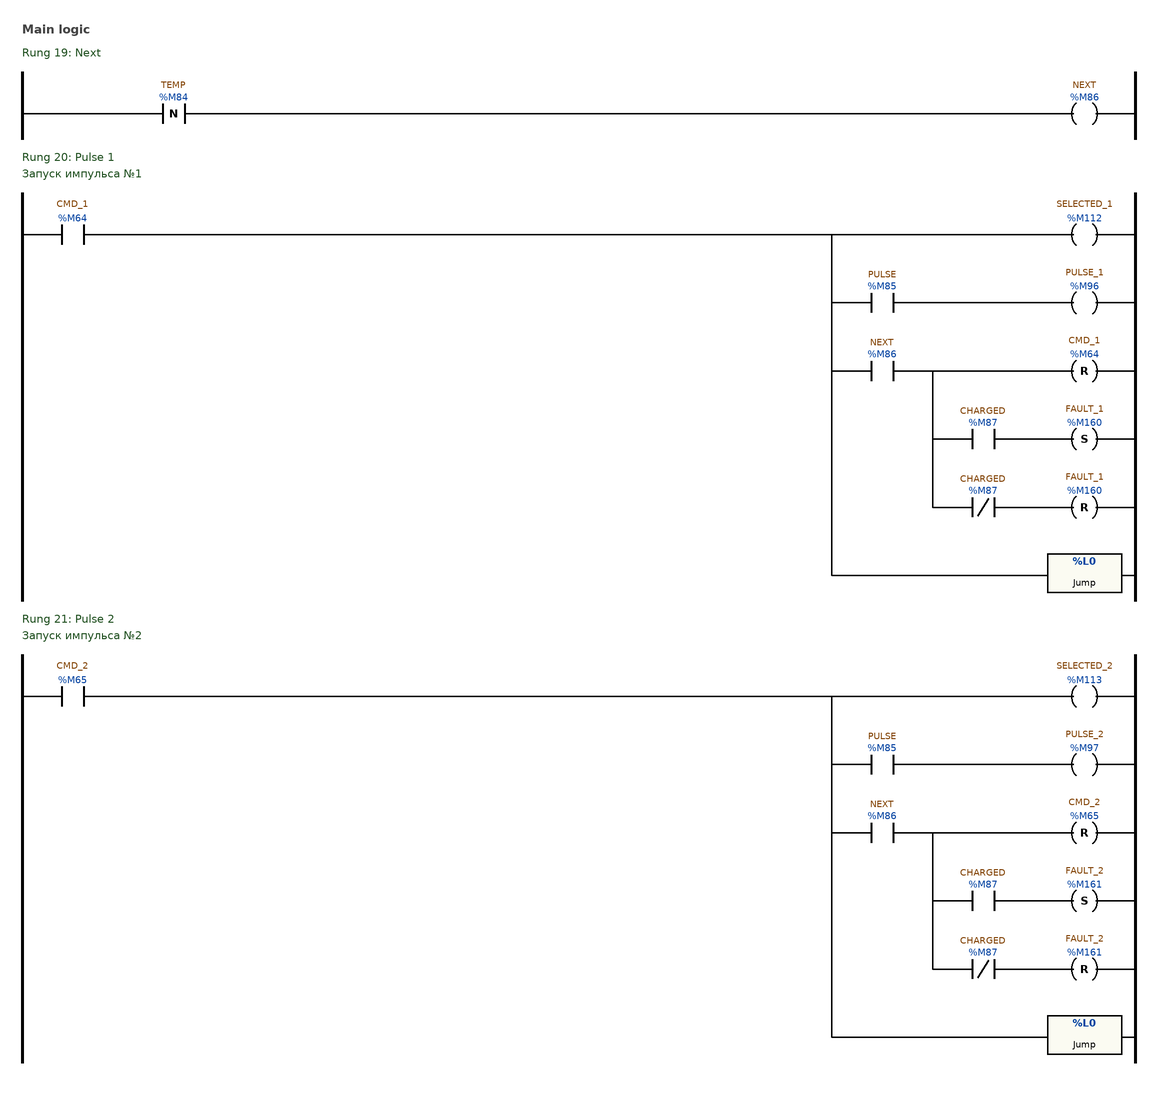

// Rung 19: Next
  LDF %M84                (* TEMP *)
  ST %M86                 (* NEXT *)
  // as ST:
  //   NEXT := FALLING(TEMP);

// Rung 20: Pulse 1
// Запуск импульса №1
  LD %M64                 (* CMD_1 *)
  MPS
  ST %M112                (* SELECTED_1 *)
  MRD
  AND %M85                (* PULSE *)
  ST %M96                 (* PULSE_1 *)
  MRD
  AND %M86                (* NEXT *)
  MPS
  R %M64                  (* CMD_1 *)
  MRD
  AND %M87                (* CHARGED *)
  S %M160                 (* FAULT_1 *)
  MPP
  ANDN %M87               (* CHARGED *)
  R %M160                 (* FAULT_1 *)
  MPP
  JMPC %L0
  // as ST:
  //   SELECTED_1 := CMD_1;
  //   PULSE_1 := CMD_1 AND PULSE;
  //   _t1 := CMD_1;
  //   _t2 := CMD_1 AND NEXT;
  //   IF _t2 THEN CMD_1 := FALSE; END_IF;
  //   IF _t2 AND CHARGED THEN FAULT_1 := TRUE; END_IF;
  //   IF _t2 AND NOT CHARGED THEN FAULT_1 := FALSE; END_IF;
  //   IF _t1 THEN JMP %L0; END_IF;

// Rung 21: Pulse 2
// Запуск импульса №2
  LD %M65                 (* CMD_2 *)
  MPS
  ST %M113                (* SELECTED_2 *)
  MRD
  AND %M85                (* PULSE *)
  ST %M97                 (* PULSE_2 *)
  MRD
  AND %M86                (* NEXT *)
  MPS
  R %M65                  (* CMD_2 *)
  MRD
  AND %M87                (* CHARGED *)
  S %M161                 (* FAULT_2 *)
  MPP
  ANDN %M87               (* CHARGED *)
  R %M161                 (* FAULT_2 *)
  MPP
  JMPC %L0
  // as ST:
  //   SELECTED_2 := CMD_2;
  //   PULSE_2 := CMD_2 AND PULSE;
  //   _t1 := CMD_2;
  //   _t2 := CMD_2 AND NEXT;
  //   IF _t2 THEN CMD_2 := FALSE; END_IF;
  //   IF _t2 AND CHARGED THEN FAULT_2 := TRUE; END_IF;
  //   IF _t2 AND NOT CHARGED THEN FAULT_2 := FALSE; END_IF;
  //   IF _t1 THEN JMP %L0; END_IF;

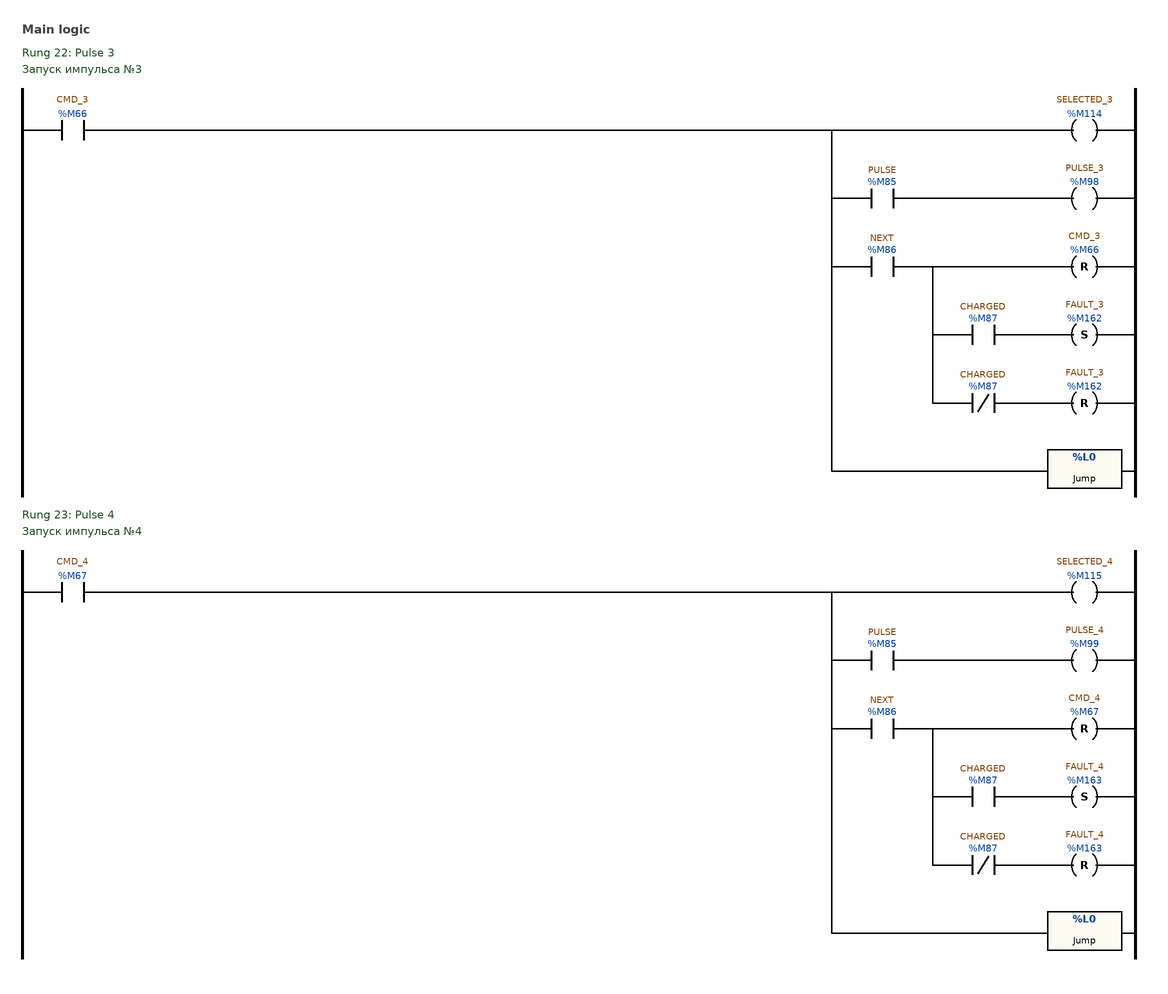

// Rung 22: Pulse 3
// Запуск импульса №3
  LD %M66                 (* CMD_3 *)
  MPS
  ST %M114                (* SELECTED_3 *)
  MRD
  AND %M85                (* PULSE *)
  ST %M98                 (* PULSE_3 *)
  MRD
  AND %M86                (* NEXT *)
  MPS
  R %M66                  (* CMD_3 *)
  MRD
  AND %M87                (* CHARGED *)
  S %M162                 (* FAULT_3 *)
  MPP
  ANDN %M87               (* CHARGED *)
  R %M162                 (* FAULT_3 *)
  MPP
  JMPC %L0
  // as ST:
  //   SELECTED_3 := CMD_3;
  //   PULSE_3 := CMD_3 AND PULSE;
  //   _t1 := CMD_3;
  //   _t2 := CMD_3 AND NEXT;
  //   IF _t2 THEN CMD_3 := FALSE; END_IF;
  //   IF _t2 AND CHARGED THEN FAULT_3 := TRUE; END_IF;
  //   IF _t2 AND NOT CHARGED THEN FAULT_3 := FALSE; END_IF;
  //   IF _t1 THEN JMP %L0; END_IF;

// Rung 23: Pulse 4
// Запуск импульса №4
  LD %M67                 (* CMD_4 *)
  MPS
  ST %M115                (* SELECTED_4 *)
  MRD
  AND %M85                (* PULSE *)
  ST %M99                 (* PULSE_4 *)
  MRD
  AND %M86                (* NEXT *)
  MPS
  R %M67                  (* CMD_4 *)
  MRD
  AND %M87                (* CHARGED *)
  S %M163                 (* FAULT_4 *)
  MPP
  ANDN %M87               (* CHARGED *)
  R %M163                 (* FAULT_4 *)
  MPP
  JMPC %L0
  // as ST:
  //   SELECTED_4 := CMD_4;
  //   PULSE_4 := CMD_4 AND PULSE;
  //   _t1 := CMD_4;
  //   _t2 := CMD_4 AND NEXT;
  //   IF _t2 THEN CMD_4 := FALSE; END_IF;
  //   IF _t2 AND CHARGED THEN FAULT_4 := TRUE; END_IF;
  //   IF _t2 AND NOT CHARGED THEN FAULT_4 := FALSE; END_IF;
  //   IF _t1 THEN JMP %L0; END_IF;

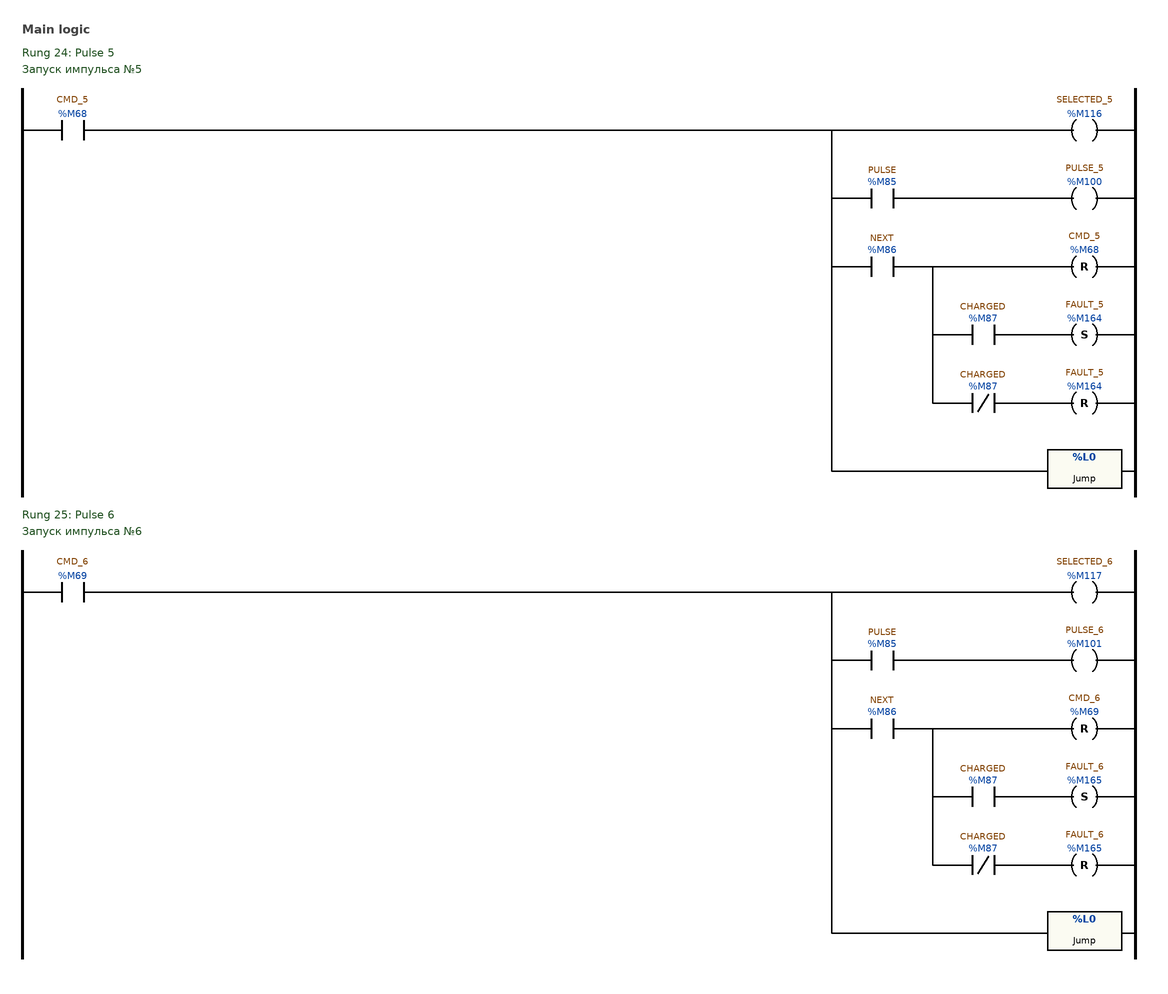

// Rung 24: Pulse 5
// Запуск импульса №5
  LD %M68                 (* CMD_5 *)
  MPS
  ST %M116                (* SELECTED_5 *)
  MRD
  AND %M85                (* PULSE *)
  ST %M100                (* PULSE_5 *)
  MRD
  AND %M86                (* NEXT *)
  MPS
  R %M68                  (* CMD_5 *)
  MRD
  AND %M87                (* CHARGED *)
  S %M164                 (* FAULT_5 *)
  MPP
  ANDN %M87               (* CHARGED *)
  R %M164                 (* FAULT_5 *)
  MPP
  JMPC %L0
  // as ST:
  //   SELECTED_5 := CMD_5;
  //   PULSE_5 := CMD_5 AND PULSE;
  //   _t1 := CMD_5;
  //   _t2 := CMD_5 AND NEXT;
  //   IF _t2 THEN CMD_5 := FALSE; END_IF;
  //   IF _t2 AND CHARGED THEN FAULT_5 := TRUE; END_IF;
  //   IF _t2 AND NOT CHARGED THEN FAULT_5 := FALSE; END_IF;
  //   IF _t1 THEN JMP %L0; END_IF;

// Rung 25: Pulse 6
// Запуск импульса №6
  LD %M69                 (* CMD_6 *)
  MPS
  ST %M117                (* SELECTED_6 *)
  MRD
  AND %M85                (* PULSE *)
  ST %M101                (* PULSE_6 *)
  MRD
  AND %M86                (* NEXT *)
  MPS
  R %M69                  (* CMD_6 *)
  MRD
  AND %M87                (* CHARGED *)
  S %M165                 (* FAULT_6 *)
  MPP
  ANDN %M87               (* CHARGED *)
  R %M165                 (* FAULT_6 *)
  MPP
  JMPC %L0
  // as ST:
  //   SELECTED_6 := CMD_6;
  //   PULSE_6 := CMD_6 AND PULSE;
  //   _t1 := CMD_6;
  //   _t2 := CMD_6 AND NEXT;
  //   IF _t2 THEN CMD_6 := FALSE; END_IF;
  //   IF _t2 AND CHARGED THEN FAULT_6 := TRUE; END_IF;
  //   IF _t2 AND NOT CHARGED THEN FAULT_6 := FALSE; END_IF;
  //   IF _t1 THEN JMP %L0; END_IF;

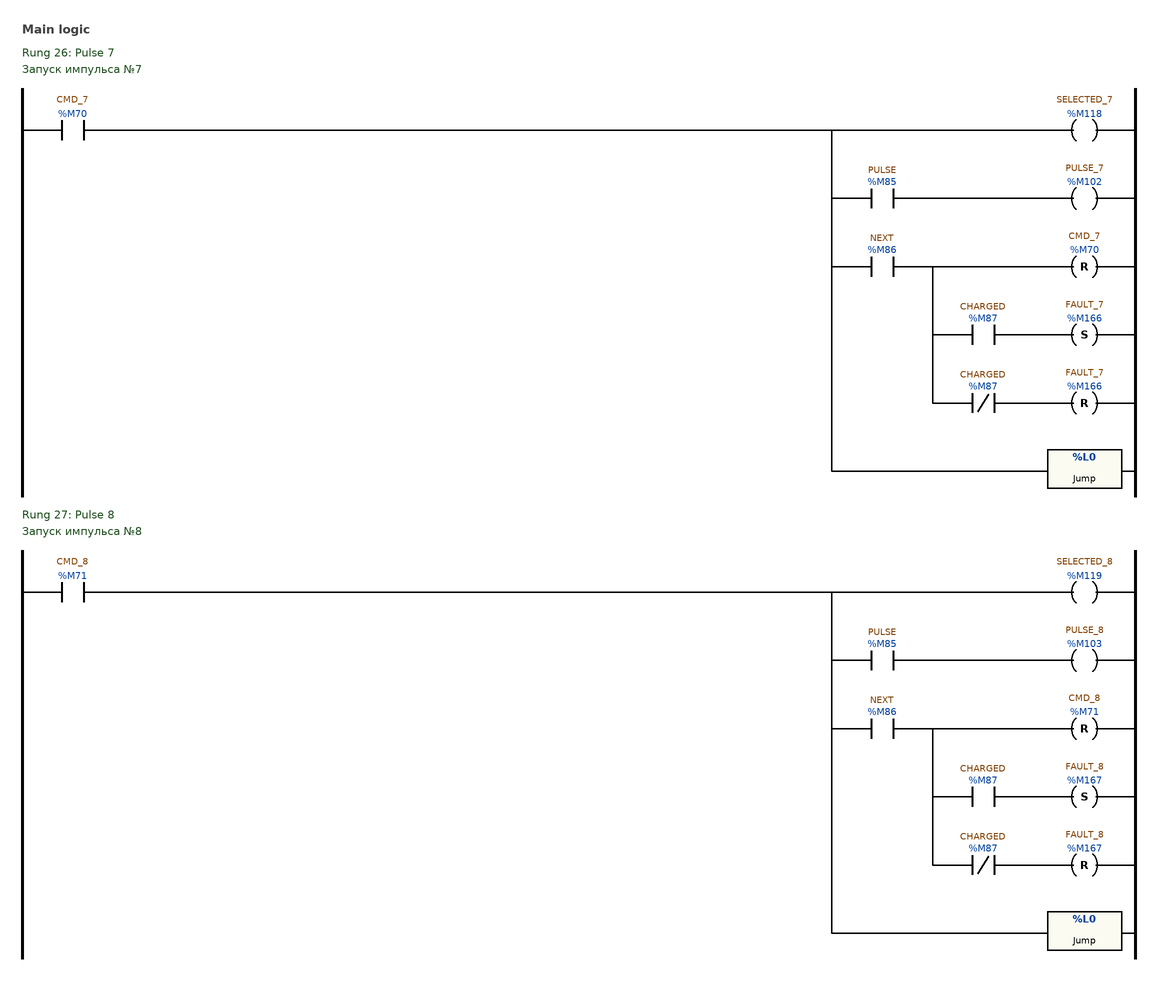

// Rung 26: Pulse 7
// Запуск импульса №7
  LD %M70                 (* CMD_7 *)
  MPS
  ST %M118                (* SELECTED_7 *)
  MRD
  AND %M85                (* PULSE *)
  ST %M102                (* PULSE_7 *)
  MRD
  AND %M86                (* NEXT *)
  MPS
  R %M70                  (* CMD_7 *)
  MRD
  AND %M87                (* CHARGED *)
  S %M166                 (* FAULT_7 *)
  MPP
  ANDN %M87               (* CHARGED *)
  R %M166                 (* FAULT_7 *)
  MPP
  JMPC %L0
  // as ST:
  //   SELECTED_7 := CMD_7;
  //   PULSE_7 := CMD_7 AND PULSE;
  //   _t1 := CMD_7;
  //   _t2 := CMD_7 AND NEXT;
  //   IF _t2 THEN CMD_7 := FALSE; END_IF;
  //   IF _t2 AND CHARGED THEN FAULT_7 := TRUE; END_IF;
  //   IF _t2 AND NOT CHARGED THEN FAULT_7 := FALSE; END_IF;
  //   IF _t1 THEN JMP %L0; END_IF;

// Rung 27: Pulse 8
// Запуск импульса №8
  LD %M71                 (* CMD_8 *)
  MPS
  ST %M119                (* SELECTED_8 *)
  MRD
  AND %M85                (* PULSE *)
  ST %M103                (* PULSE_8 *)
  MRD
  AND %M86                (* NEXT *)
  MPS
  R %M71                  (* CMD_8 *)
  MRD
  AND %M87                (* CHARGED *)
  S %M167                 (* FAULT_8 *)
  MPP
  ANDN %M87               (* CHARGED *)
  R %M167                 (* FAULT_8 *)
  MPP
  JMPC %L0
  // as ST:
  //   SELECTED_8 := CMD_8;
  //   PULSE_8 := CMD_8 AND PULSE;
  //   _t1 := CMD_8;
  //   _t2 := CMD_8 AND NEXT;
  //   IF _t2 THEN CMD_8 := FALSE; END_IF;
  //   IF _t2 AND CHARGED THEN FAULT_8 := TRUE; END_IF;
  //   IF _t2 AND NOT CHARGED THEN FAULT_8 := FALSE; END_IF;
  //   IF _t1 THEN JMP %L0; END_IF;

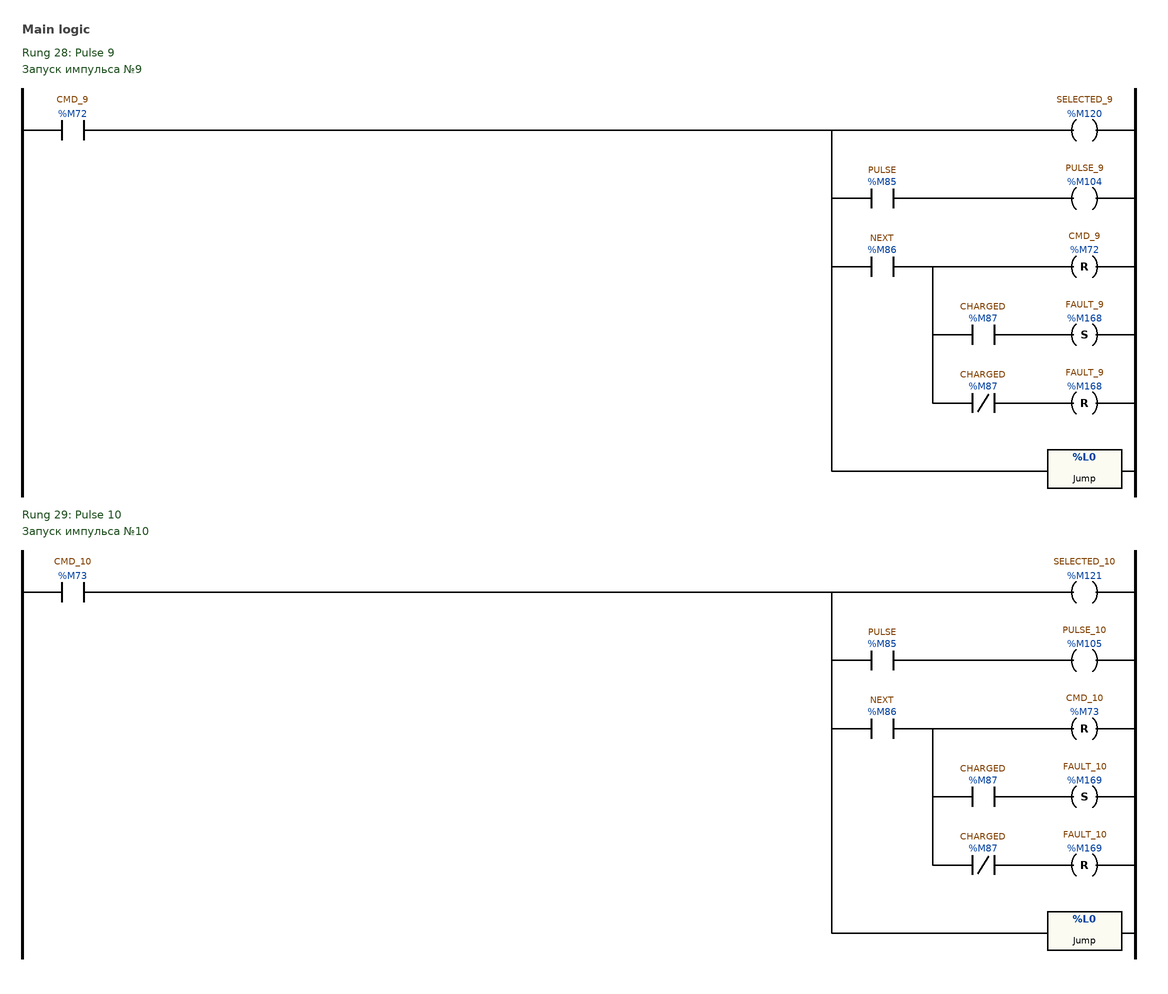

// Rung 28: Pulse 9
// Запуск импульса №9
  LD %M72                 (* CMD_9 *)
  MPS
  ST %M120                (* SELECTED_9 *)
  MRD
  AND %M85                (* PULSE *)
  ST %M104                (* PULSE_9 *)
  MRD
  AND %M86                (* NEXT *)
  MPS
  R %M72                  (* CMD_9 *)
  MRD
  AND %M87                (* CHARGED *)
  S %M168                 (* FAULT_9 *)
  MPP
  ANDN %M87               (* CHARGED *)
  R %M168                 (* FAULT_9 *)
  MPP
  JMPC %L0
  // as ST:
  //   SELECTED_9 := CMD_9;
  //   PULSE_9 := CMD_9 AND PULSE;
  //   _t1 := CMD_9;
  //   _t2 := CMD_9 AND NEXT;
  //   IF _t2 THEN CMD_9 := FALSE; END_IF;
  //   IF _t2 AND CHARGED THEN FAULT_9 := TRUE; END_IF;
  //   IF _t2 AND NOT CHARGED THEN FAULT_9 := FALSE; END_IF;
  //   IF _t1 THEN JMP %L0; END_IF;

// Rung 29: Pulse 10
// Запуск импульса №10
  LD %M73                 (* CMD_10 *)
  MPS
  ST %M121                (* SELECTED_10 *)
  MRD
  AND %M85                (* PULSE *)
  ST %M105                (* PULSE_10 *)
  MRD
  AND %M86                (* NEXT *)
  MPS
  R %M73                  (* CMD_10 *)
  MRD
  AND %M87                (* CHARGED *)
  S %M169                 (* FAULT_10 *)
  MPP
  ANDN %M87               (* CHARGED *)
  R %M169                 (* FAULT_10 *)
  MPP
  JMPC %L0
  // as ST:
  //   SELECTED_10 := CMD_10;
  //   PULSE_10 := CMD_10 AND PULSE;
  //   _t1 := CMD_10;
  //   _t2 := CMD_10 AND NEXT;
  //   IF _t2 THEN CMD_10 := FALSE; END_IF;
  //   IF _t2 AND CHARGED THEN FAULT_10 := TRUE; END_IF;
  //   IF _t2 AND NOT CHARGED THEN FAULT_10 := FALSE; END_IF;
  //   IF _t1 THEN JMP %L0; END_IF;

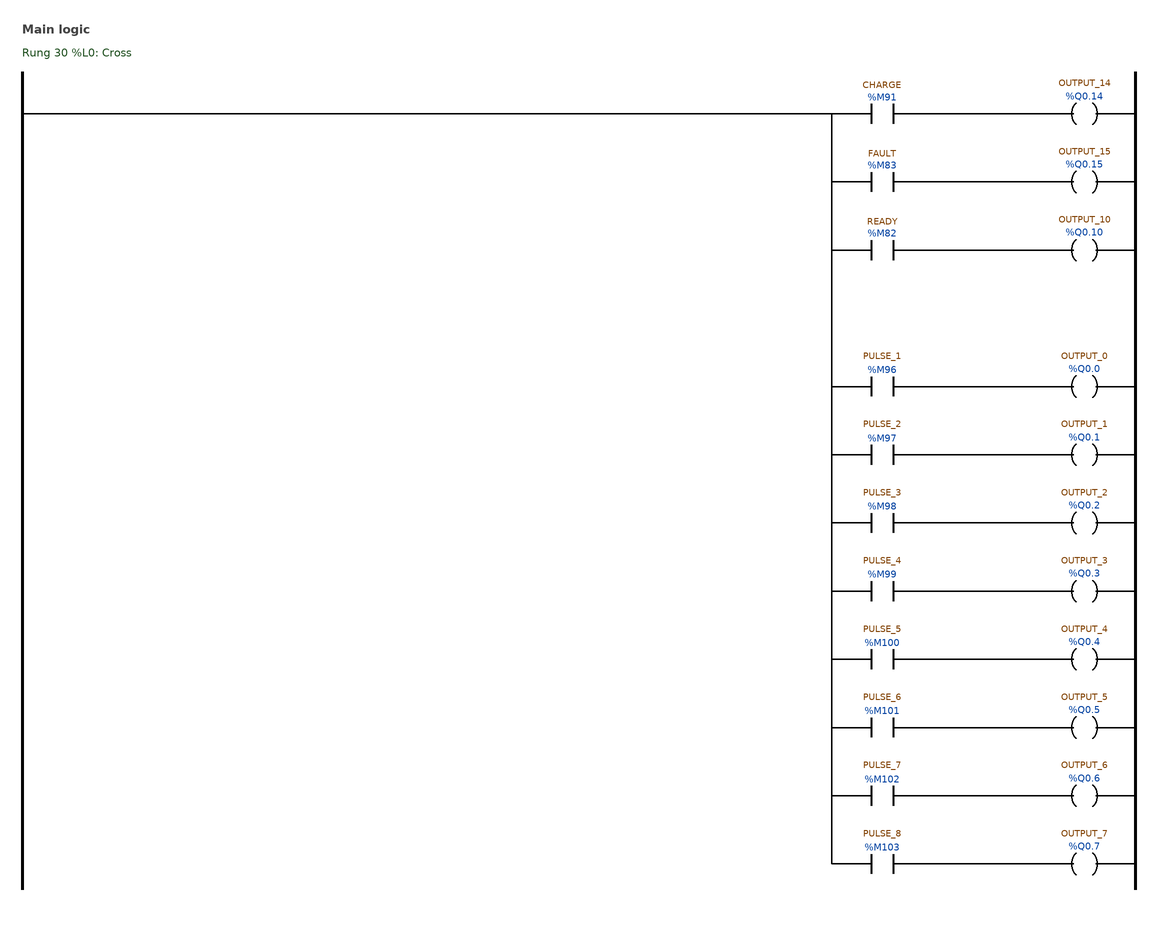

// Rung 30 %L0: Cross
  %L0:
  LD 1
  MPS
  AND %M91                (* CHARGE *)
  ST %Q0.14               (* OUTPUT_14 *)
  MRD
  AND %M83                (* FAULT *)
  ST %Q0.15               (* OUTPUT_15 *)
  MRD
  AND %M82                (* READY *)
  ST %Q0.10               (* OUTPUT_10 *)
  MRD
  AND %M96                (* PULSE_1 *)
  ST %Q0.0                (* OUTPUT_0 *)
  MRD
  AND %M97                (* PULSE_2 *)
  ST %Q0.1                (* OUTPUT_1 *)
  MRD
  AND %M98                (* PULSE_3 *)
  ST %Q0.2                (* OUTPUT_2 *)
  MRD
  AND %M99                (* PULSE_4 *)
  ST %Q0.3                (* OUTPUT_3 *)
  MRD
  AND %M100               (* PULSE_5 *)
  ST %Q0.4                (* OUTPUT_4 *)
  MRD
  AND %M101               (* PULSE_6 *)
  ST %Q0.5                (* OUTPUT_5 *)
  MRD
  AND %M102               (* PULSE_7 *)
  ST %Q0.6                (* OUTPUT_6 *)
  MPP
  AND %M103               (* PULSE_8 *)
  ST %Q0.7                (* OUTPUT_7 *)
  // as ST:
  //   %L0:
  //   OUTPUT_14 := CHARGE;
  //   OUTPUT_15 := FAULT;
  //   OUTPUT_10 := READY;
  //   OUTPUT_0 := PULSE_1;
  //   OUTPUT_1 := PULSE_2;
  //   OUTPUT_2 := PULSE_3;
  //   OUTPUT_3 := PULSE_4;
  //   OUTPUT_4 := PULSE_5;
  //   OUTPUT_5 := PULSE_6;
  //   OUTPUT_6 := PULSE_7;
  //   OUTPUT_7 := PULSE_8;
